{attribute 'linkalways'} 
{attribute 'no_explicit_call' := 'This FB is a CLASS and must be accessed using methods or properties'}
{attribute 'enable_dynamic_creation'}
FUNCTION_BLOCK ABSTRACT StructuredDatatypeBase EXTENDS DatatypeBase IMPLEMENTS I_StructuredDatatype
VAR
	membersHost : MembersHost;
END_VAR

METHOD PUBLIC Accept
VAR_INPUT
	Visitor : I_DatatypeVisitor;
END_VAR
Visitor.VisitDatatype(THIS^);
membersHost.Accept(Visitor);
END_METHOD

METHOD PROTECTED AddMember
VAR_INPUT
	MemberName : T_MAXSTRING;
	Member : I_Datatype;
END_VAR
membersHost.AddMember(MemberName, Member);
END_METHOD

METHOD PUBLIC GetMemberEnumerator : I_KeyValueForwardEnumerator
VAR_INPUT
END_VAR
GetMemberEnumerator := membersHost.GetMemberEnumerator();
END_METHOD

PROPERTY PUBLIC ABSTRACT Identifier : T_MAXSTRING
GET
END_GET
END_PROPERTY

PROPERTY PUBLIC IecType : T_MAXSTRING
GET
IecType := 'STRUCT';
END_GET
END_PROPERTY

METHOD PUBLIC SerializeTypeWith
VAR_INPUT
	Serializer : I_Serializer;
END_VAR
Serializer.StartObject();
Serializer.AddKeyString('name',Identifier);
Serializer.AddKeyString('type',IecType);	
membersHost.SerializeTypeWith(Serializer);
Serializer.EndObject();
END_METHOD

METHOD PUBLIC SerializeWith
VAR_INPUT
	Serializer : I_Serializer;
END_VAR
Serializer.StartObject();
membersHost.SerializeWith(Serializer);
Serializer.EndObject();
END_METHOD

METHOD PUBLIC TryCopy : BOOL
VAR_INPUT
	Source : I_Datatype;
END_VAR
VAR
	SourceAsStructure : I_StructuredDatatype;
END_VAR
IF NOT Source.TryResolveAsStructuredType(SourceAsStructure) THEN
	RETURN;
END_IF

IF SourceAsStructure.Identifier <> Identifier THEN
	RETURN;
END_IF

memcpy(Address, Source.Address, Size);
END_METHOD

METHOD TryDeserializeFrom : BOOL
VAR_INPUT
	Deserializer : I_Deserializer;
	Feedback : I_DeserializerFeedback;
END_VAR
TryDeserializeFrom := membersHost.TryDeserializeFrom(Deserializer, Feedback);
END_METHOD

METHOD PUBLIC TryGetMemberByName : BOOL
VAR_INPUT
	Name : T_MAXSTRING;
	Destination : REFERENCE TO I_Datatype;
END_VAR
VAR
	member : I_Datatype;
END_VAR
IF NOT membersHost.TryGetMemberByName(Name, member) THEN 
	RETURN;
END_IF

Destination := member;
TryGetMemberByName := TRUE;
END_METHOD

METHOD PUBLIC TryResolveAsStructuredType : BOOL
VAR_INPUT
	Destination : REFERENCE TO I_StructuredDatatype;
END_VAR
Destination := THIS^;
TryResolveAsStructuredType := TRUE;
END_METHOD

END_FUNCTION_BLOCK

(* stored: Version 1.1.0.1, ProductVersion 3.1.4024.12
   POU StructuredDatatypeBase: Id {d625e009-5f55-02c3-36d6-363c53933949}, SpecialFunc None
   Folder Protected: Id {7be81008-5185-0ecf-2c87-21a945dccc6c}
   Method Accept: Id {06765757-4f9c-06e9-3ba8-c4dbd62f08c0}
   Method AddMember: Id {000f5fe3-c73b-0a5c-3784-f4147181b91f}
   Method GetMemberEnumerator: Id {fac9ada8-4cb2-073e-22b0-6df830bd06b4}
   Property Identifier: Id {fad1b093-141e-0c94-3cbf-d2814230ee8f}
   Get Get: Id {0ba07a67-9506-0b52-2c39-54987f0097d7}
   Property IecType: Id {a8c18764-bb60-0e02-27e9-99f1e4f4ba10}
   Get Get: Id {bc004734-b432-0c60-2e2e-c258a8f38112}
   Method SerializeTypeWith: Id {9654791f-6cce-4be3-aa2e-1642f4102f87}
   Method SerializeWith: Id {f673cce2-1a3e-44bc-81da-e8bc2c037902}
   Method TryCopy: Id {2a52ab7e-c04c-4dca-9c5a-bd85f10678c4}
   Method TryDeserializeFrom: Id {59671805-cc69-411a-a0b1-4ff94095acb6}
   Method TryGetMemberByName: Id {8f166c4e-7a97-0c21-3753-3c2e46dcf112}
   Method TryResolveAsStructuredType: Id {4cf287f6-cc3a-0aaf-0d50-e2dcf54e34fd} *)
